// TIA Portal V21 export
TYPE "LBC_typeAnalogScaleConfiguration"
TITLE = LBC_typeAnalogScaleConfiguration
// Module related configuration parameters
   STRUCT
      referenceDesignator { S7_SetPoint := 'True'} : WString[25] := WSTRING#'AnalogScale';   // Device name or device ID
      physicalUnitInput { S7_SetPoint := 'True'} : String[10] := 'unit';   // Physical unit (like [°C], [kWh], etc.) for the input value
      physicalUnitOutput { S7_SetPoint := 'True'} : String[10] := 'unit';   // Physical unit (like [°C], [kWh], etc.) for the output value
      default { S7_SetPoint := 'True'} : LReal := 0.0;   // Default OUTPUT value to be returned if function block is not enabled or quality is bad
      inputValueMax { S7_SetPoint := 'True'} : LReal := 100.0;   // Maximum limit of the process value
      inputValueMin { S7_SetPoint := 'True'} : LReal := -100.0;   // Minimum limit of the process value
      scaleInputUppPoint { S7_SetPoint := 'True'} : LReal := 100.0;   // Upper point for the process value
      scaleInputLowPoint { S7_SetPoint := 'True'} : LReal := -100.0;   // Lower point for the process value
      scaleOutputUppPoint { S7_SetPoint := 'True'} : LReal := 200.0;   // Upper point for the analog process output
      scaleOutputLowPoint { S7_SetPoint := 'True'} : LReal := -200.0;   // Lower point for the analog process output
      disableAlarms { S7_SetPoint := 'True'} : Bool;   // Disable the alarms of the block
   END_STRUCT;
END_TYPE
